FUNCTION Convert_USINT_TO_INT : BOOL
VAR_INPUT
	in : USINT;
	out : REFERENCE TO INT;
END_VAR
VAR
	converted : INT;
END_VAR

converted := USINT_TO_INT(in);

IF (INT_TO_USINT(converted) <> in) THEN
	RETURN;
END_IF

out := converted;
Convert_USINT_TO_INT := TRUE;

END_FUNCTION

(* stored: Version 1.1.0.1, ProductVersion 3.1.4024.12
   POU Convert_USINT_TO_INT: Id {edc2918f-44d8-469b-9549-76bad91ba009}, SpecialFunc None *)
